(* Logix 5000 project; controller Stepper_Driver_3401L_SUB vendor 1 type 14 code 155 rev 20.12; software revision 20.01 *)

TASK MainTask (continuous, watchdog 500 ms) : MainProgram

MODULES
   Local : vendor 1 type 14 code 155 (PointIO 0, rev 20.12)
       : vendor 10 type 150 code 185 (PointIO 5, rev 1.1, Output RPI 50 ms)
           Local:5:I.DATA2.14   // 3401L Module OK Bit
           Local:5:I.DATA2.13   // 3401L Configuration Error Bit
           Local:5:I.DATA2.10   // 3401L position invalid bit
           Local:5:I.DATA2.0   // CW Move In Progress
           Local:5:I.DATA2.1   // CCW Move In Progress
           Local:5:I.DATA2.7   // Move Complete
           Local:5:I.DATA2.15   // Config Mode 1=config 0=command
       : 1734-IE2V (PointIO 2, rev 3.1, Input RPI 80 ms)
      Discrete_IO : Embedded (PointIO 1, rev 20.11, Output RPI 20 ms)
       : vendor 1 type 109 code 13 (PointIO 4, rev 3.1, Output RPI 80 ms)
       : 1734-OE2V (PointIO 3, rev 3.1, Output RPI 80 ms)
END_MODULES

PROGRAM MainProgram   (* main routine MainRoutine *)
VAR
   Abs_Move : INT[8] := ([0] := 1, [3] := 500, [4] := 1, [6] := 25, [7] := 25);
        [0]   // Abs Move
        [3]   // 1s place
        [4]   // 1000
        [5]   // speed
        [6]   // acc
        [7]   // dec
        [2]   // 1000th place
   Configuration_3401L : INT[8] := ([0] := -32592, [3] := 5); {constant}
   distance : INT := -10500;
   Incr_Move : INT[8] := ([0] := 2, [2] := -10, [3] := -500, [4] := 1, [5] := 500, [6] := 10, [7] := 10);
        [2]   // distance (x1000's) +
        [7]   // dec 10
        [0]   // Incr Move
        [6]   // acc 10
        [3]   // + distance (x1)
        [4]   // speed (x1000's) +
        [5]   // + speed (x1)
   M_State : INT := 1;
   one_shot_1 : BOOL;
   one_shot_2 : BOOL := 1;
   one_shot_M : BOOL;
   Position : DINT := -10500;
   Preset_3401L : INT[8] := ([0] := 512); {constant}
   Preset_Reset_Move_Complete : INT[8] := ([0] := 512, [2] := 209);
   Reset_Errors_3401 : INT[8] := ([0] := 2048); {constant}
   s1 : INT;
   Speed : DINT := 1500;
   state : INT := 1;
   Stepper_Move : INT[8] := ([0] := 2, [2] := -10, [3] := -500, [4] := 1, [5] := 500, [6] := 10, [7] := 10);
        [6]   // Acc
        [0]   // Move type
        [2]   // 1000th place
        [3]   // 1s place pos
        [4]   // 1000th place
        [5]   // 1s place speed
        [7]   // Dec
   Subready : BOOL;
   SubState0 : BOOL;
   SubState1 : BOOL;
   t1 : TIMER := (PRE := 500);
   t2 : TIMER := (PRE := 500);
   t3 : TIMER := (PRE := 500);
   t4 : TIMER := (PRE := 500);
   t5 : TIMER := (PRE := 500);
   t6 : TIMER := (PRE := 500);
   t7 : TIMER := (PRE := 500);
   t8 : TIMER := (PRE := 500);
END_VAR

ROUTINE CalculatePositionSpeed   (* structured text *)
   //
   //
   sbr();
   
   	Position := distance;
   
   	// position
   	Incr_Move[2]:= Position / 1000; 				// MSW integer divide
   	Incr_Move[3]:= Position - (Incr_Move[2] * 1000); // LSW remainder
   	// speed
   	//
   	Incr_Move[4]:= Speed / 1000; 				// MSW integer divide
   	Incr_Move[5]:= Speed - (Incr_Move[4] * 1000); // LSW remainder
   //
   ret();
END_ROUTINE

ROUTINE MainRoutine   (* ladder *)
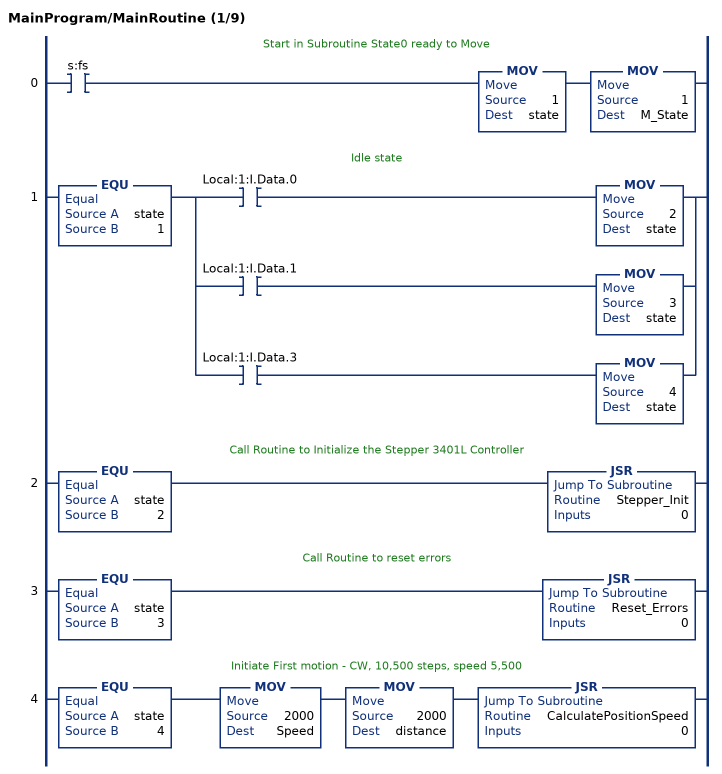
   // Start in Subroutine State0 ready to Move
   0: XIC(s:fs)MOV(1,state)MOV(1,M_State);
   // Idle state
   1: EQU(state,1)[XIC(Local:1:I.Data.0) MOV(2,state) ,[XIC(Local:1:I.Data.1) MOV(3,state) ,XIC(Local:1:I.Data.3) MOV(4,state) ] ];
   // Call Routine to Initialize the Stepper 3401L Controller
   2: EQU(state,2)JSR(Stepper_Init,0);
   // Call Routine to reset errors
   3: EQU(state,3)JSR(Reset_Errors,0);
   // Initiate First motion - CW, 10,500 steps, speed 5,500
   4: EQU(state,4)MOV(2000,Speed)MOV(2000,distance)JSR(CalculatePositionSpeed,0);
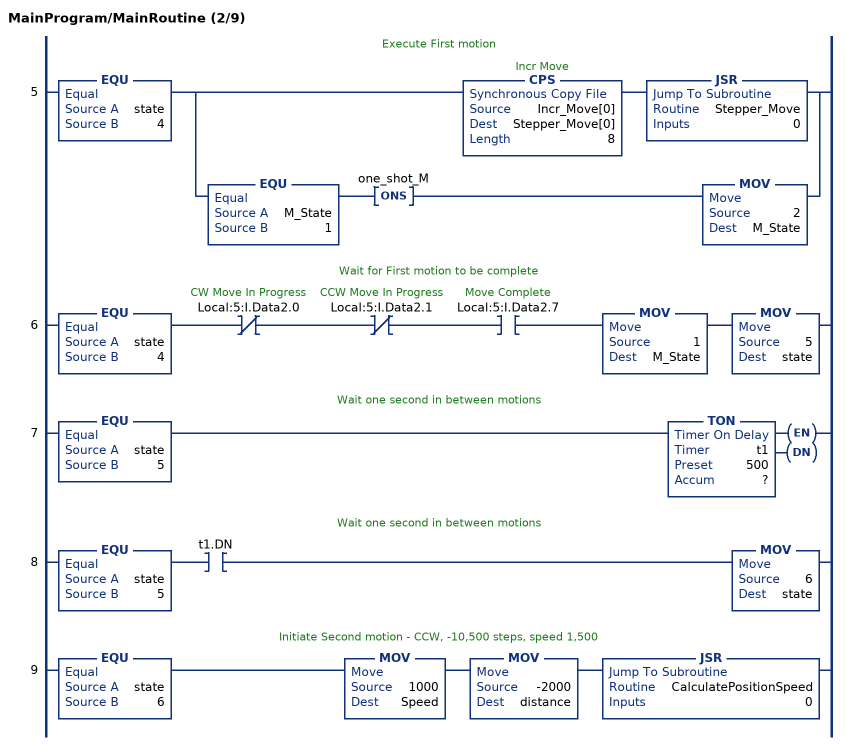
   // Execute First motion
   5: EQU(state,4)[CPS(Incr_Move[0],Stepper_Move[0],8) JSR(Stepper_Move,0) ,EQU(M_State,1) ONS(one_shot_M) MOV(2,M_State) ];
   // Wait for First motion to be complete
   6: EQU(state,4)XIO(Local:5:I.Data2.0)XIO(Local:5:I.Data2.1)XIC(Local:5:I.Data2.7)MOV(1,M_State)MOV(5,state);
   // Wait one second in between motions
   7: EQU(state,5)TON(t1,?,?);
   // Wait one second in between motions
   8: EQU(state,5)XIC(t1.DN)MOV(6,state);
   // Initiate Second motion - CCW, -10,500 steps, speed 1,500
   9: EQU(state,6)MOV(1000,Speed)MOV(-2000,distance)JSR(CalculatePositionSpeed,0);
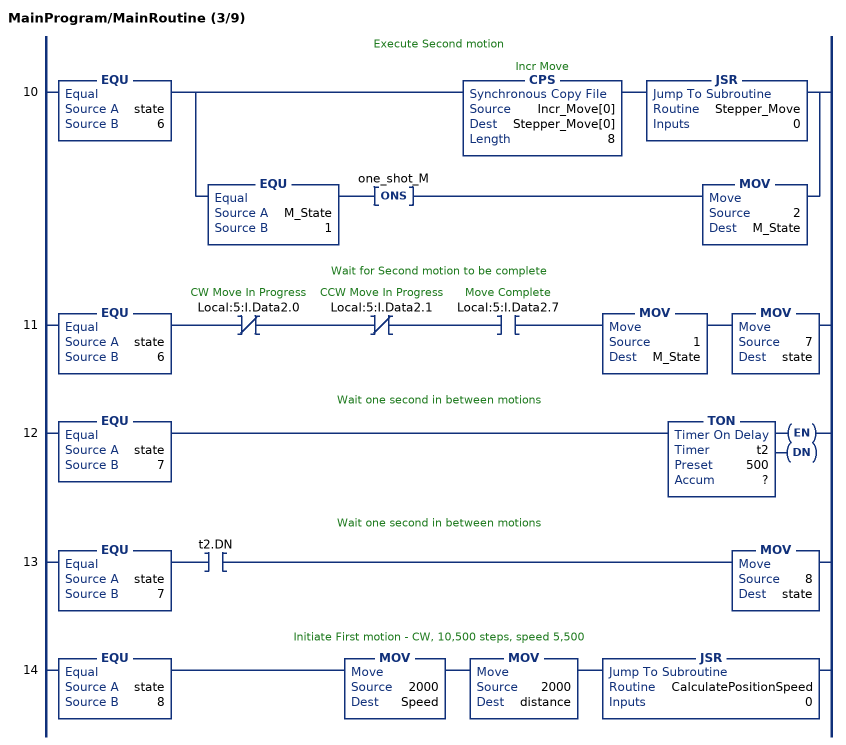
   // Execute Second motion
   10: EQU(state,6)[CPS(Incr_Move[0],Stepper_Move[0],8) JSR(Stepper_Move,0) ,EQU(M_State,1) ONS(one_shot_M) MOV(2,M_State) ];
   // Wait for Second motion to be complete
   11: EQU(state,6)XIO(Local:5:I.Data2.0)XIO(Local:5:I.Data2.1)XIC(Local:5:I.Data2.7)MOV(1,M_State)MOV(7,state);
   // Wait one second in between motions
   12: EQU(state,7)TON(t2,?,?);
   // Wait one second in between motions
   13: EQU(state,7)XIC(t2.DN)MOV(8,state);
   // Initiate First motion - CW, 10,500 steps, speed 5,500
   14: EQU(state,8)MOV(2000,Speed)MOV(2000,distance)JSR(CalculatePositionSpeed,0);
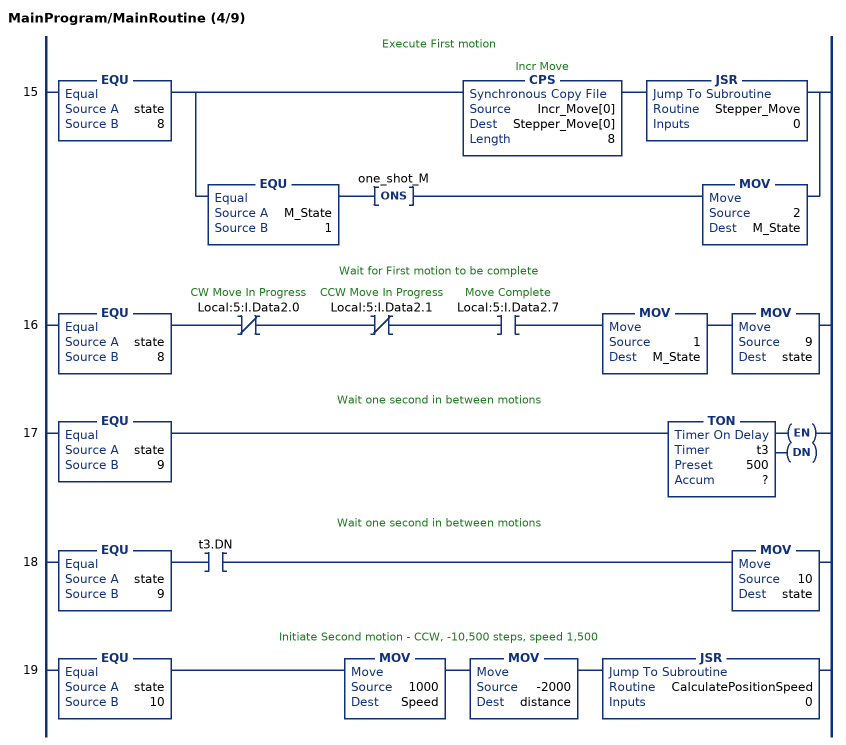
   // Execute First motion
   15: EQU(state,8)[CPS(Incr_Move[0],Stepper_Move[0],8) JSR(Stepper_Move,0) ,EQU(M_State,1) ONS(one_shot_M) MOV(2,M_State) ];
   // Wait for First motion to be complete
   16: EQU(state,8)XIO(Local:5:I.Data2.0)XIO(Local:5:I.Data2.1)XIC(Local:5:I.Data2.7)MOV(1,M_State)MOV(9,state);
   // Wait one second in between motions
   17: EQU(state,9)TON(t3,?,?);
   // Wait one second in between motions
   18: EQU(state,9)XIC(t3.DN)MOV(10,state);
   // Initiate Second motion - CCW, -10,500 steps, speed 1,500
   19: EQU(state,10)MOV(1000,Speed)MOV(-2000,distance)JSR(CalculatePositionSpeed,0);
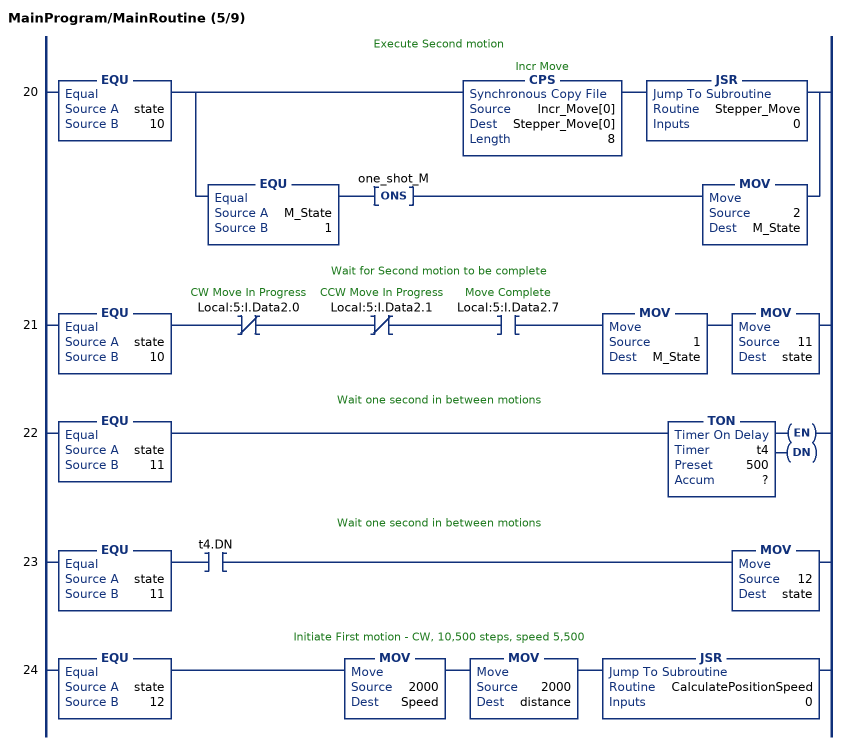
   // Execute Second motion
   20: EQU(state,10)[CPS(Incr_Move[0],Stepper_Move[0],8) JSR(Stepper_Move,0) ,EQU(M_State,1) ONS(one_shot_M) MOV(2,M_State) ];
   // Wait for Second motion to be complete
   21: EQU(state,10)XIO(Local:5:I.Data2.0)XIO(Local:5:I.Data2.1)XIC(Local:5:I.Data2.7)MOV(1,M_State)MOV(11,state);
   // Wait one second in between motions
   22: EQU(state,11)TON(t4,?,?);
   // Wait one second in between motions
   23: EQU(state,11)XIC(t4.DN)MOV(12,state);
   // Initiate First motion - CW, 10,500 steps, speed 5,500
   24: EQU(state,12)MOV(2000,Speed)MOV(2000,distance)JSR(CalculatePositionSpeed,0);
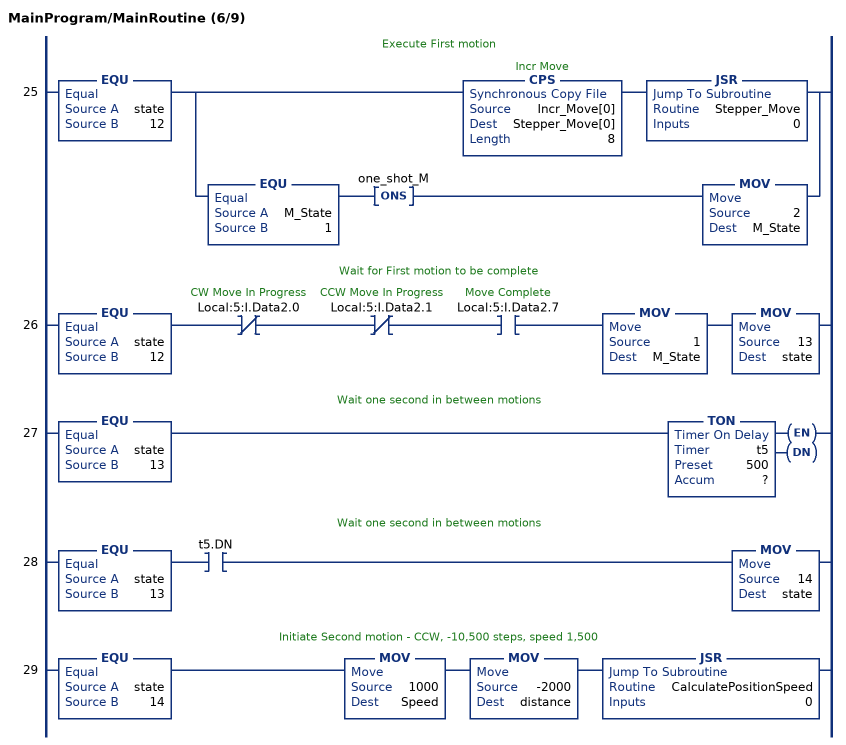
   // Execute First motion
   25: EQU(state,12)[CPS(Incr_Move[0],Stepper_Move[0],8) JSR(Stepper_Move,0) ,EQU(M_State,1) ONS(one_shot_M) MOV(2,M_State) ];
   // Wait for First motion to be complete
   26: EQU(state,12)XIO(Local:5:I.Data2.0)XIO(Local:5:I.Data2.1)XIC(Local:5:I.Data2.7)MOV(1,M_State)MOV(13,state);
   // Wait one second in between motions
   27: EQU(state,13)TON(t5,?,?);
   // Wait one second in between motions
   28: EQU(state,13)XIC(t5.DN)MOV(14,state);
   // Initiate Second motion - CCW, -10,500 steps, speed 1,500
   29: EQU(state,14)MOV(1000,Speed)MOV(-2000,distance)JSR(CalculatePositionSpeed,0);
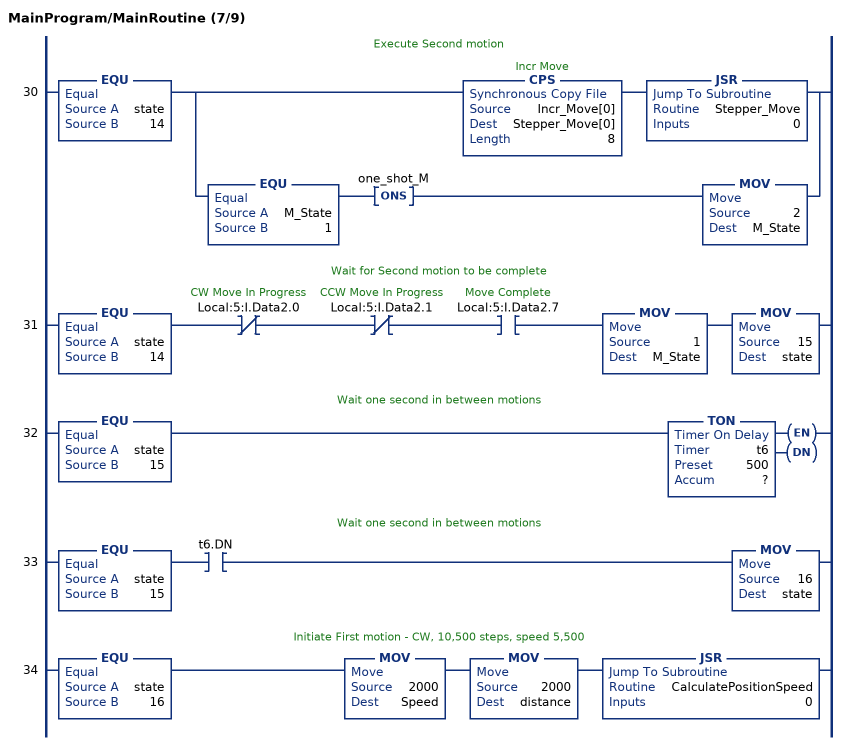
   // Execute Second motion
   30: EQU(state,14)[CPS(Incr_Move[0],Stepper_Move[0],8) JSR(Stepper_Move,0) ,EQU(M_State,1) ONS(one_shot_M) MOV(2,M_State) ];
   // Wait for Second motion to be complete
   31: EQU(state,14)XIO(Local:5:I.Data2.0)XIO(Local:5:I.Data2.1)XIC(Local:5:I.Data2.7)MOV(1,M_State)MOV(15,state);
   // Wait one second in between motions
   32: EQU(state,15)TON(t6,?,?);
   // Wait one second in between motions
   33: EQU(state,15)XIC(t6.DN)MOV(16,state);
   // Initiate First motion - CW, 10,500 steps, speed 5,500
   34: EQU(state,16)MOV(2000,Speed)MOV(2000,distance)JSR(CalculatePositionSpeed,0);
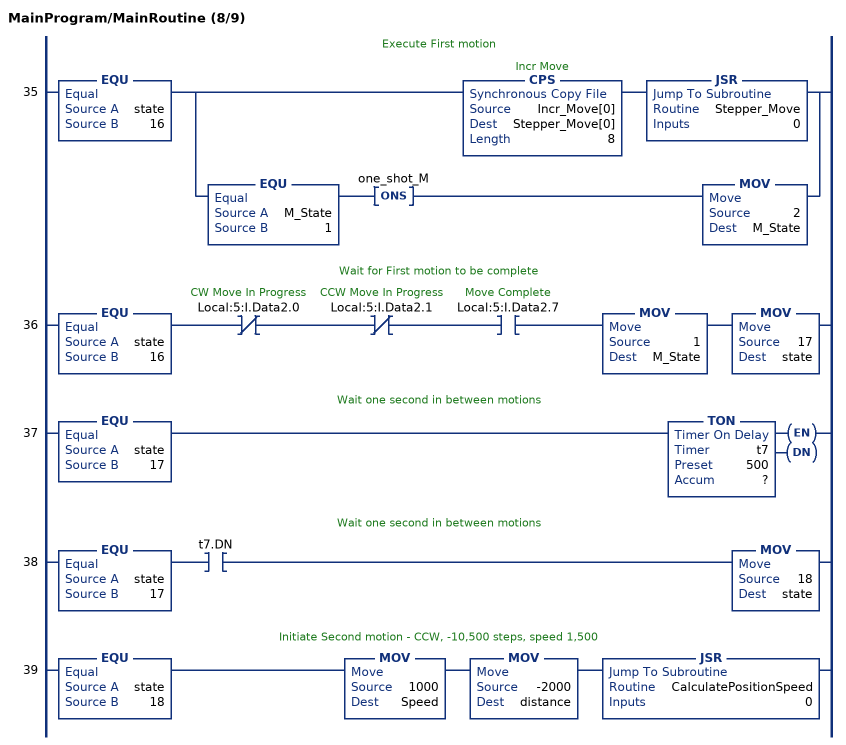
   // Execute First motion
   35: EQU(state,16)[CPS(Incr_Move[0],Stepper_Move[0],8) JSR(Stepper_Move,0) ,EQU(M_State,1) ONS(one_shot_M) MOV(2,M_State) ];
   // Wait for First motion to be complete
   36: EQU(state,16)XIO(Local:5:I.Data2.0)XIO(Local:5:I.Data2.1)XIC(Local:5:I.Data2.7)MOV(1,M_State)MOV(17,state);
   // Wait one second in between motions
   37: EQU(state,17)TON(t7,?,?);
   // Wait one second in between motions
   38: EQU(state,17)XIC(t7.DN)MOV(18,state);
   // Initiate Second motion - CCW, -10,500 steps, speed 1,500
   39: EQU(state,18)MOV(1000,Speed)MOV(-2000,distance)JSR(CalculatePositionSpeed,0);
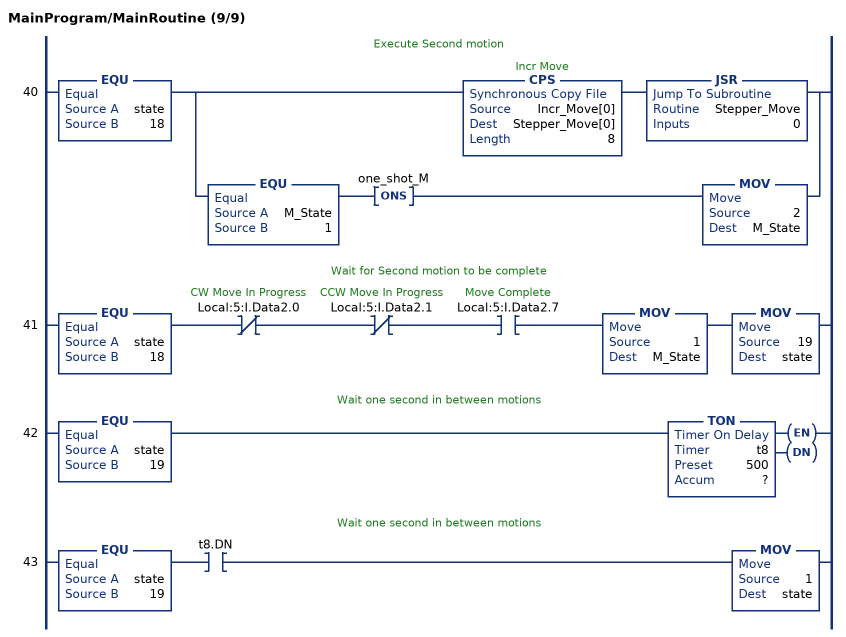
   // Execute Second motion
   40: EQU(state,18)[CPS(Incr_Move[0],Stepper_Move[0],8) JSR(Stepper_Move,0) ,EQU(M_State,1) ONS(one_shot_M) MOV(2,M_State) ];
   // Wait for Second motion to be complete
   41: EQU(state,18)XIO(Local:5:I.Data2.0)XIO(Local:5:I.Data2.1)XIC(Local:5:I.Data2.7)MOV(1,M_State)MOV(19,state);
   // Wait one second in between motions
   42: EQU(state,19)TON(t8,?,?);
   // Wait one second in between motions
   43: EQU(state,19)XIC(t8.DN)MOV(1,state);
END_ROUTINE

ROUTINE Reset_Errors   (* ladder *)
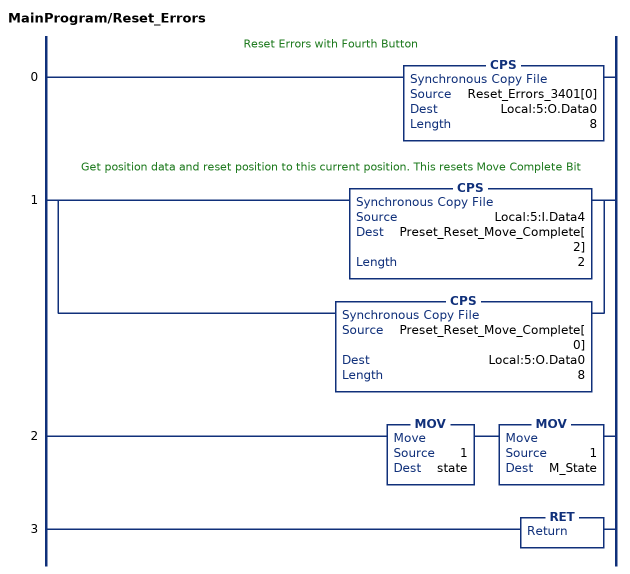
   // Reset Errors with Fourth Button
   0: CPS(Reset_Errors_3401[0],Local:5:O.Data0,8);
   // Get position data and reset position to this current position. This resets Move Complete Bit
   1: [CPS(Local:5:I.Data4,Preset_Reset_Move_Complete[2],2) ,CPS(Preset_Reset_Move_Complete[0],Local:5:O.Data0,8) ];
   2: MOV(1,state)MOV(1,M_State);
   3: RET();
END_ROUTINE

ROUTINE Stepper_Init   (* ladder *)
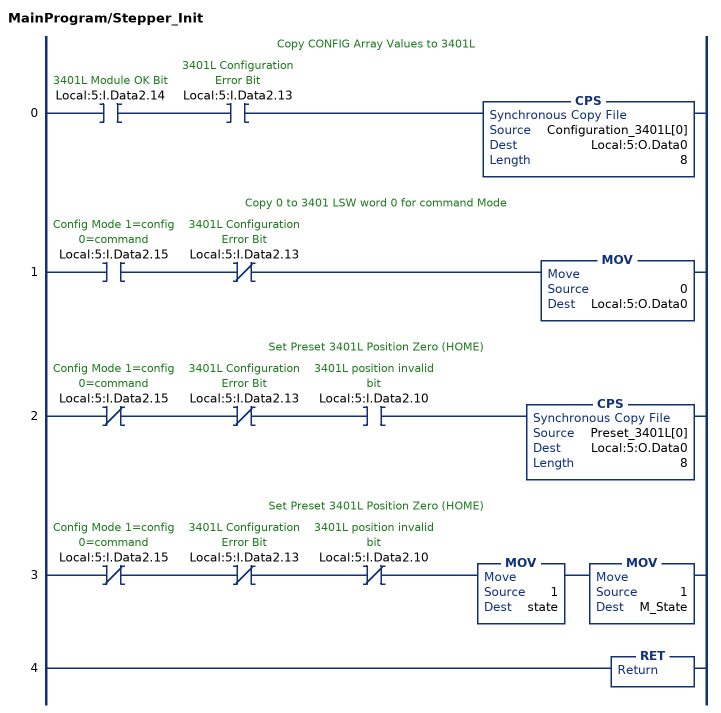
   // Copy CONFIG Array Values to 3401L
   0: XIC(Local:5:I.Data2.14)XIC(Local:5:I.Data2.13)CPS(Configuration_3401L[0],Local:5:O.Data0,8);
   // Copy 0 to 3401 LSW word 0 for command Mode
   1: XIC(Local:5:I.Data2.15)XIO(Local:5:I.Data2.13)MOV(0,Local:5:O.Data0);
   // Set Preset 3401L Position Zero (HOME)
   2: XIO(Local:5:I.Data2.15)XIO(Local:5:I.Data2.13)XIC(Local:5:I.Data2.10)CPS(Preset_3401L[0],Local:5:O.Data0,8);
   // Set Preset 3401L Position Zero (HOME)
   3: XIO(Local:5:I.Data2.15)XIO(Local:5:I.Data2.13)XIO(Local:5:I.Data2.10)MOV(1,state)MOV(1,M_State);
   4: RET();
END_ROUTINE

ROUTINE Stepper_Move   (* ladder *)
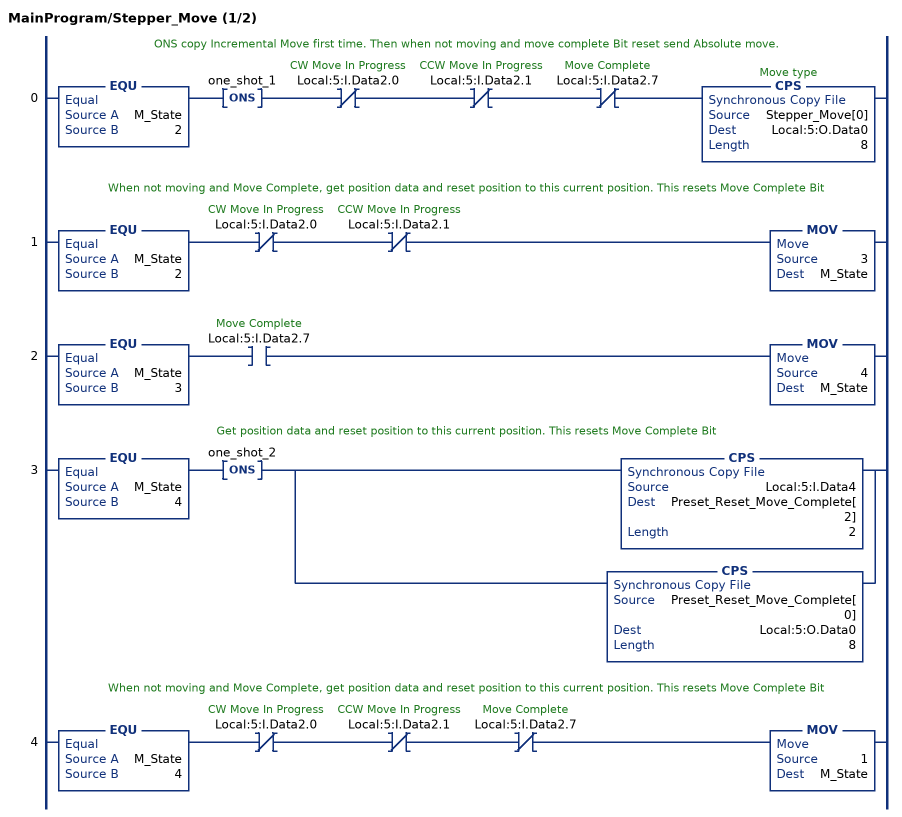
   // ONS copy Incremental Move first time. Then when not moving and move complete Bit reset send Absolute move.
   0: EQU(M_State,2)ONS(one_shot_1)XIO(Local:5:I.Data2.0)XIO(Local:5:I.Data2.1)XIO(Local:5:I.Data2.7)CPS(Stepper_Move[0],Local:5:O.Data0,8);
   // When not moving and Move Complete, get position data and reset position to this current position. This resets Move Complete Bit
   1: EQU(M_State,2)XIO(Local:5:I.Data2.0)XIO(Local:5:I.Data2.1)MOV(3,M_State);
   2: EQU(M_State,3)XIC(Local:5:I.Data2.7)MOV(4,M_State);
   // Get position data and reset position to this current position. This resets Move Complete Bit
   3: EQU(M_State,4)ONS(one_shot_2)[CPS(Local:5:I.Data4,Preset_Reset_Move_Complete[2],2) ,CPS(Preset_Reset_Move_Complete[0],Local:5:O.Data0,8) ];
   // When not moving and Move Complete, get position data and reset position to this current position. This resets Move Complete Bit
   4: EQU(M_State,4)XIO(Local:5:I.Data2.0)XIO(Local:5:I.Data2.1)XIO(Local:5:I.Data2.7)MOV(1,M_State);
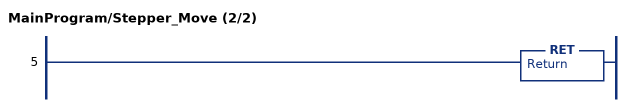
   5: RET();
END_ROUTINE
END_PROGRAM
